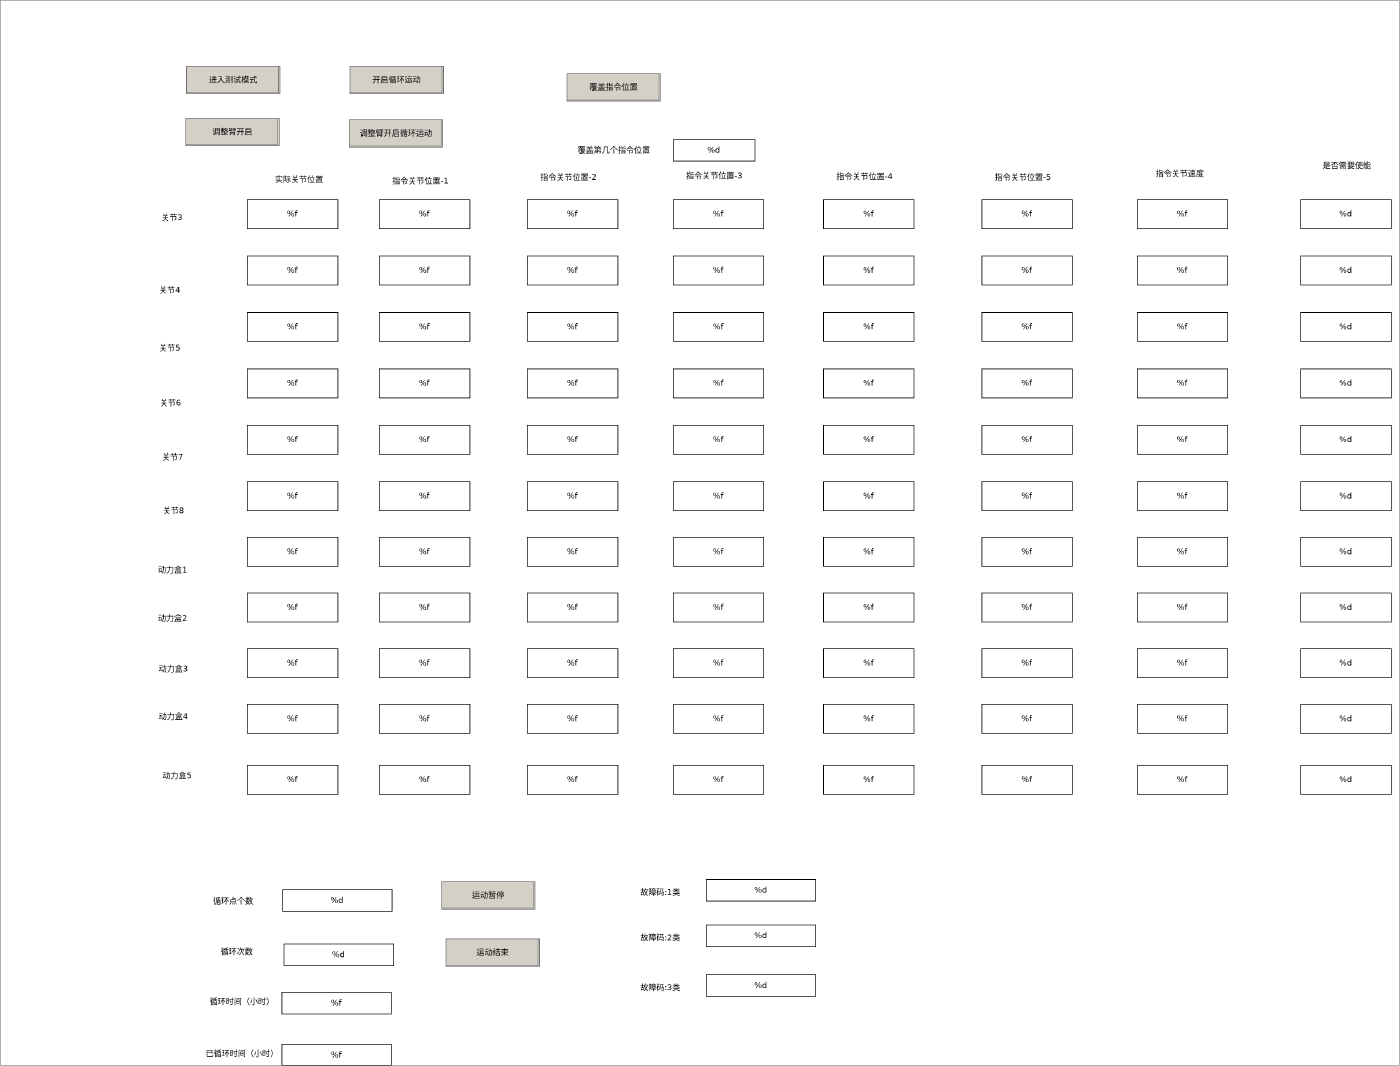
VISUALIZATION cycle_a4  // 1910x1455
    Button (254,90 128x38), "进入测试模式", colour toggle: g_cycleTest.m_enterCycleTestMode[4]
        toggle g_cycleTest.m_enterCycleTestMode[4]
    Button (477,90 128x38), "开启循环运动", colour toggle: g_cycleTest.m_startMotion[4]
        toggle g_cycleTest.m_startMotion[4]
    Label (501,233 145x28), "指令关节位置-1"
    Label (333,230 150x30), "实际关节位置"
    Rectangle (337,503 124x40), "%f", text variable: g_cycleTest.m_actJntPos[4][1]
    Label (162,283 145x28), "关节3"
    Label (159,382 145x28), "关节4"
    Label (159,461 145x28), "关节5"
    Label (160,536 145x28), "关节6"
    Label (163,610 145x28), "关节7"
    Label (164,683 145x28), "关节8"
    Label (163,764 145x28), "动力盒1"
    Label (163,830 145x28), "动力盒2"
    Label (169,1045 145x28), "动力盒5"
    Label (164,899 145x28), "动力盒3"
    Label (164,964 145x28), "动力盒4"
    Rectangle (337,580 124x40), "%f", text variable: g_cycleTest.m_actJntPos[4][2]
    Rectangle (337,657 124x40), "%f", text variable: g_cycleTest.m_actJntPos[4][3]
    Rectangle (337,733 124x40), "%f", text variable: g_cycleTest.m_actJntPos[4][4]
    Rectangle (337,809 124x40), "%f", text variable: g_cycleTest.m_actJntPos[4][5]
    Rectangle (337,885 124x40), "%f", text variable: g_cycleTest.m_actJntPos[4][6]
    Rectangle (337,961 124x40), "%f", text variable: g_cycleTest.m_actJntPos[4][7]
    Rectangle (337,1044 124x40), "%f", text variable: g_cycleTest.m_actJntPos[4][8]
    Rectangle (337,272 124x40), "%f", text variable: g_cycleTest.m_actJntPosSetup[4][3]
    Rectangle (337,349 124x40), "%f", text variable: g_cycleTest.m_actJntPosSetup[4][4]
    Rectangle (337,426 124x40), "%f", text variable: g_cycleTest.m_actJntPosSetup[4][5]
    Rectangle (517,272 124x40), "%f", text variable: g_cycleTest.m_targetJntPosSetup[4,1][3]
        OnMouseClick: write the text variable via Default
    Rectangle (517,349 124x40), "%f", text variable: g_cycleTest.m_targetJntPosSetup[4,1][4]
        OnMouseClick: write the text variable via Default
    Rectangle (517,426 124x40), "%f", text variable: g_cycleTest.m_targetJntPosSetup[4,1][5]
        OnMouseClick: write the text variable via Default
    Rectangle (517,503 124x40), "%f", text variable: g_cycleTest.m_targetJntPos[4,1][1]
        OnMouseClick: write the text variable via Default
    Rectangle (517,580 124x40), "%f", text variable: g_cycleTest.m_targetJntPos[4,1][2]
        OnMouseClick: write the text variable via Default
    Rectangle (517,657 124x40), "%f", text variable: g_cycleTest.m_targetJntPos[4,1][3]
        OnMouseClick: write the text variable via Default
    Rectangle (517,733 124x40), "%f", text variable: g_cycleTest.m_targetJntPos[4,1][4]
        OnMouseClick: write the text variable via Default
    Rectangle (517,809 124x40), "%f", text variable: g_cycleTest.m_targetJntPos[4,1][5]
        OnMouseClick: write the text variable via Default
    Rectangle (517,885 124x40), "%f", text variable: g_cycleTest.m_targetJntPos[4,1][6]
        OnMouseClick: write the text variable via Default
    Rectangle (517,961 124x40), "%f", text variable: g_cycleTest.m_targetJntPos[4,1][7]
        OnMouseClick: write the text variable via Default
    Rectangle (517,1044 124x40), "%f", text variable: g_cycleTest.m_targetJntPos[4,1][8]
        OnMouseClick: write the text variable via Default
    Label (703,228 145x28), "指令关节位置-2"
    Rectangle (719,272 124x40), "%f", text variable: g_cycleTest.m_targetJntPosSetup[4,2][3]
        OnMouseClick: write the text variable via Default
    Rectangle (719,349 124x40), "%f", text variable: g_cycleTest.m_targetJntPosSetup[4,2][4]
        OnMouseClick: write the text variable via Default
    Rectangle (719,426 124x40), "%f", text variable: g_cycleTest.m_targetJntPosSetup[4,2][5]
        OnMouseClick: write the text variable via Default
    Rectangle (719,503 124x40), "%f", text variable: g_cycleTest.m_targetJntPos[4,2][1]
        OnMouseClick: write the text variable via Default
    Rectangle (719,580 124x40), "%f", text variable: g_cycleTest.m_targetJntPos[4,2][2]
        OnMouseClick: write the text variable via Default
    Rectangle (719,657 124x40), "%f", text variable: g_cycleTest.m_targetJntPos[4,2][3]
        OnMouseClick: write the text variable via Default
    Rectangle (719,733 124x40), "%f", text variable: g_cycleTest.m_targetJntPos[4,2][4]
        OnMouseClick: write the text variable via Default
    Rectangle (719,809 124x40), "%f", text variable: g_cycleTest.m_targetJntPos[4,2][5]
        OnMouseClick: write the text variable via Default
    Rectangle (719,885 124x40), "%f", text variable: g_cycleTest.m_targetJntPos[4,2][6]
        OnMouseClick: write the text variable via Default
    Rectangle (719,961 124x40), "%f", text variable: g_cycleTest.m_targetJntPos[4,2][7]
        OnMouseClick: write the text variable via Default
    Rectangle (719,1044 124x40), "%f", text variable: g_cycleTest.m_targetJntPos[4,2][8]
        OnMouseClick: write the text variable via Default
    Label (902,226 145x28), "指令关节位置-3"
    Rectangle (918,272 124x40), "%f", text variable: g_cycleTest.m_targetJntPosSetup[4,3][3]
        OnMouseClick: write the text variable via Default
    Rectangle (918,349 124x40), "%f", text variable: g_cycleTest.m_targetJntPosSetup[4,3][4]
        OnMouseClick: write the text variable via Default
    Rectangle (918,426 124x40), "%f", text variable: g_cycleTest.m_targetJntPosSetup[4,3][5]
        OnMouseClick: write the text variable via Default
    Rectangle (918,503 124x40), "%f", text variable: g_cycleTest.m_targetJntPos[4,3][1]
        OnMouseClick: write the text variable via Default
    Rectangle (918,580 124x40), "%f", text variable: g_cycleTest.m_targetJntPos[4,3][2]
        OnMouseClick: write the text variable via Default
    Rectangle (918,657 124x40), "%f", text variable: g_cycleTest.m_targetJntPos[4,3][3]
        OnMouseClick: write the text variable via Default
    Rectangle (918,733 124x40), "%f", text variable: g_cycleTest.m_targetJntPos[4,3][4]
        OnMouseClick: write the text variable via Default
    Rectangle (918,809 124x40), "%f", text variable: g_cycleTest.m_targetJntPos[4,3][5]
        OnMouseClick: write the text variable via Default
    Rectangle (918,885 124x40), "%f", text variable: g_cycleTest.m_targetJntPos[4,3][6]
        OnMouseClick: write the text variable via Default
    Rectangle (918,961 124x40), "%f", text variable: g_cycleTest.m_targetJntPos[4,3][7]
        OnMouseClick: write the text variable via Default
    Rectangle (918,1044 124x40), "%f", text variable: g_cycleTest.m_targetJntPos[4,3][8]
        OnMouseClick: write the text variable via Default
    Label (1107,227 145x28), "指令关节位置-4"
    Rectangle (1123,272 124x40), "%f", text variable: g_cycleTest.m_targetJntPosSetup[4,4][3]
        OnMouseClick: write the text variable via Default
    Rectangle (1123,349 124x40), "%f", text variable: g_cycleTest.m_targetJntPosSetup[4,4][4]
        OnMouseClick: write the text variable via Default
    Rectangle (1123,426 124x40), "%f", text variable: g_cycleTest.m_targetJntPosSetup[4,4][5]
        OnMouseClick: write the text variable via Default
    Rectangle (1123,503 124x40), "%f", text variable: g_cycleTest.m_targetJntPos[4,4][1]
        OnMouseClick: write the text variable via Default
    Rectangle (1123,580 124x40), "%f", text variable: g_cycleTest.m_targetJntPos[4,4][2]
        OnMouseClick: write the text variable via Default
    Rectangle (1123,657 124x40), "%f", text variable: g_cycleTest.m_targetJntPos[4,4][3]
        OnMouseClick: write the text variable via Default
    Rectangle (1123,733 124x40), "%f", text variable: g_cycleTest.m_targetJntPos[4,4][4]
        OnMouseClick: write the text variable via Default
    Rectangle (1123,809 124x40), "%f", text variable: g_cycleTest.m_targetJntPos[4,4][5]
        OnMouseClick: write the text variable via Default
    Rectangle (1123,885 124x40), "%f", text variable: g_cycleTest.m_targetJntPos[4,4][6]
        OnMouseClick: write the text variable via Default
    Rectangle (1123,961 124x40), "%f", text variable: g_cycleTest.m_targetJntPos[4,4][7]
        OnMouseClick: write the text variable via Default
    Rectangle (1123,1044 124x40), "%f", text variable: g_cycleTest.m_targetJntPos[4,4][8]
        OnMouseClick: write the text variable via Default
    Label (1323,228 145x28), "指令关节位置-5"
    Rectangle (1339,272 124x40), "%f", text variable: g_cycleTest.m_targetJntPosSetup[4,5][3]
        OnMouseClick: write the text variable via Default
    Rectangle (1339,349 124x40), "%f", text variable: g_cycleTest.m_targetJntPosSetup[4,5][4]
        OnMouseClick: write the text variable via Default
    Rectangle (1339,426 124x40), "%f", text variable: g_cycleTest.m_targetJntPosSetup[4,5][5]
        OnMouseClick: write the text variable via Default
    Rectangle (1339,503 124x40), "%f", text variable: g_cycleTest.m_targetJntPos[4,5][1]
        OnMouseClick: write the text variable via Default
    Rectangle (1339,580 124x40), "%f", text variable: g_cycleTest.m_targetJntPos[4,5][2]
        OnMouseClick: write the text variable via Default
    Rectangle (1339,657 124x40), "%f", text variable: g_cycleTest.m_targetJntPos[4,5][3]
        OnMouseClick: write the text variable via Default
    Rectangle (1339,733 124x40), "%f", text variable: g_cycleTest.m_targetJntPos[4,5][4]
        OnMouseClick: write the text variable via Default
    Rectangle (1339,809 124x40), "%f", text variable: g_cycleTest.m_targetJntPos[4,5][5]
        OnMouseClick: write the text variable via Default
    Rectangle (1339,885 124x40), "%f", text variable: g_cycleTest.m_targetJntPos[4,5][6]
        OnMouseClick: write the text variable via Default
    Rectangle (1339,961 124x40), "%f", text variable: g_cycleTest.m_targetJntPos[4,5][7]
        OnMouseClick: write the text variable via Default
    Rectangle (1339,1044 124x40), "%f", text variable: g_cycleTest.m_targetJntPos[4,5][8]
        OnMouseClick: write the text variable via Default
    Button (253,161 128x38), "调整臂开启", colour toggle: g_cycleTest.m_enterCycleTestModeSetup[4]
        toggle g_cycleTest.m_enterCycleTestModeSetup[4]
    Button (476,163 128x38), "调整臂开启循环运动", colour toggle: g_cycleTest.m_startMotionSetup[4]
        toggle g_cycleTest.m_startMotionSetup[4]
    Label (1537,223 145x28), "指令关节速度"
    Rectangle (1551,272 124x40), "%f", text variable: g_cycleTest.m_targetJntVelSetup[4][3]
        OnMouseClick: write the text variable via Default
    Rectangle (1551,349 124x40), "%f", text variable: g_cycleTest.m_targetJntVelSetup[4][4]
        OnMouseClick: write the text variable via Default
    Rectangle (1551,426 124x40), "%f", text variable: g_cycleTest.m_targetJntVelSetup[4][5]
        OnMouseClick: write the text variable via Default
    Rectangle (1551,503 124x40), "%f", text variable: g_cycleTest.m_targetJntVelN8[4][1]
        OnMouseClick: write the text variable via Default
    Rectangle (1551,580 124x40), "%f", text variable: g_cycleTest.m_targetJntVelN8[4][2]
        OnMouseClick: write the text variable via Default
    Rectangle (1551,657 124x40), "%f", text variable: g_cycleTest.m_targetJntVelN8[4][3]
        OnMouseClick: write the text variable via Default
    Rectangle (1551,733 124x40), "%f", text variable: g_cycleTest.m_targetJntVelN8[4][4]
        OnMouseClick: write the text variable via Default
    Rectangle (1551,809 124x40), "%f", text variable: g_cycleTest.m_targetJntVelN8[4][5]
        OnMouseClick: write the text variable via Default
    Rectangle (1551,885 124x40), "%f", text variable: g_cycleTest.m_targetJntVelN8[4][6]
        OnMouseClick: write the text variable via Default
    Rectangle (1551,961 124x40), "%f", text variable: g_cycleTest.m_targetJntVelN8[4][7]
        OnMouseClick: write the text variable via Default
    Rectangle (1551,1044 124x40), "%f", text variable: g_cycleTest.m_targetJntVelN8[4][8]
        OnMouseClick: write the text variable via Default
    Button (773,100 128x38), "覆盖指令位置", colour toggle: g_cycleTest.m_coverCmdPos[4]
        tap g_cycleTest.m_coverCmdPos[4]
    Rectangle (918,190 112x30), "%d", text variable: g_cycleTest.m_pntIdForCoverCmd[4]
        OnMouseClick: write the text variable via Default
    Label (765,191 145x28), "覆盖第几个指令位置"
    Label (243,1215 150x30), "循环点个数"
    Rectangle (385,1214 150x30), "%d", text variable: g_cycleTest.m_pointSum[4]
        OnMouseClick: write the text variable via Default
    Rectangle (387,1288 150x30), "%d", text variable: g_cycleTest.m_curCycleNum[4]
        OnMouseClick: write the text variable via Default
    Label (248,1284 150x30), "循环次数"
    Button (602,1203 128x38), "运动暂停", colour toggle: g_cycleTest.m_pause[4]
        toggle g_cycleTest.m_pause[4]
    Button (608,1281 128x38), "运动结束", colour toggle: g_cycleTest.m_finish[4]
        tap g_cycleTest.m_finish[4]
    Rectangle (384,1354 150x30), "%f", text variable: g_cycleTest.m_tgtCycleTime[4]
        OnMouseClick: write the text variable via Default
    Label (255,1352 150x30), "循环时间（小时）"
    Rectangle (384,1425 150x30), "%f", text variable: g_cycleTest.m_curCycleTime[4]
        OnMouseClick: write the text variable via Default
    Label (255,1423 150x30), "已循环时间（小时）"
    Label (1765,211 145x30), "是否需要使能"
    Rectangle (1774,272 124x40), "%d", text variable: g_cycleTest.m_jntEnableSetup[4][3]
        OnMouseClick: write the text variable via Default
    Rectangle (1774,349 124x40), "%d", text variable: g_cycleTest.m_jntEnableSetup[4][4]
        OnMouseClick: write the text variable via Default
    Rectangle (1774,426 124x40), "%d", text variable: g_cycleTest.m_jntEnableSetup[4][5]
        OnMouseClick: write the text variable via Default
    Rectangle (1774,503 124x40), "%d", text variable: g_cycleTest.m_jntEnable[4][1]
        OnMouseClick: write the text variable via Default
    Rectangle (1774,580 124x40), "%d", text variable: g_cycleTest.m_jntEnable[4][2]
        OnMouseClick: write the text variable via Default
    Rectangle (1774,657 124x40), "%d", text variable: g_cycleTest.m_jntEnable[4][3]
        OnMouseClick: write the text variable via Default
    Rectangle (1774,733 124x40), "%d", text variable: g_cycleTest.m_jntEnable[4][4]
        OnMouseClick: write the text variable via Default
    Rectangle (1774,809 124x40), "%d", text variable: g_cycleTest.m_jntEnable[4][5]
        OnMouseClick: write the text variable via Default
    Rectangle (1774,885 124x40), "%d", text variable: g_cycleTest.m_jntEnable[4][6]
        OnMouseClick: write the text variable via Default
    Rectangle (1774,961 124x40), "%d", text variable: g_cycleTest.m_jntEnable[4][7]
        OnMouseClick: write the text variable via Default
    Rectangle (1774,1044 124x40), "%d", text variable: g_cycleTest.m_jntEnable[4][8]
        OnMouseClick: write the text variable via Default
    Rectangle (963,1200 150x30), "%d", text variable: GVL_interactUI.g_errIdType1
        OnMouseClick: write the text variable via Default
    Label (826,1203 150x30), "故障码:1类"
    Rectangle (963,1262 150x30), "%d", text variable: GVL_interactUI.g_errIdType2
        OnMouseClick: write the text variable via Default
    Label (826,1265 150x30), "故障码:2类"
    Rectangle (963,1330 150x30), "%d", text variable: GVL_interactUI.g_errIdType3
        OnMouseClick: write the text variable via Default
    Label (826,1333 150x30), "故障码:3类"
END_VISUALIZATION

(* stored: Version 1.1.0.1, ProductVersion 3.1.4024.11
   Visu cycle_a4: Id {0ab73bfb-e415-44c2-a1e5-e017427878d1} *)
